(* PLC project testproj, Beckhoff Automation GmbH TwinCAT PLC Control 3.5.20.50 *)
(* stored: creationDateTime 2025-07-01T11:02:16.1300929, modificationDateTime 2025-07-01T11:02:16.1300929 *)

FUNCTION_BLOCK AnaMon
  VAR_INPUT
    WQC : BYTE;
    OSLevel : BYTE;
    V : REAL;
    VSclMin : REAL;
    VSclMax : REAL;
    VUnit : INT;
    VAHEn : BOOL;
    VWHEn : BOOL;
    VTHEn : BOOL;
    VTLEn : BOOL;
    VWLEn : BOOL;
    VALEn : BOOL;
  END_VAR
  VAR_OUTPUT
    VAHAct : BOOL;
    VWHAct : BOOL;
    VTHAct : BOOL;
    VTLAct : BOOL;
    VWLAct : BOOL;
    VALAct : BOOL;
  END_VAR
  VAR
    VAHLim : REAL;
    VWHLim : REAL;
    VTHLim : REAL;
    VTLLim : REAL;
    VWLLim : REAL;
    VALLim : REAL;
  END_VAR

            
                
// Copy MTP base variables to local temporaries (READ access)


VAHAct := vOut >= alarmHigh;
VWHAct := vOut >= warningHigh;
VTHAct := vOut >= toleranceHigh;
VTLAct := vOut <= toleranceLow;
VWLAct := vOut <= warningLow;
VALAct := vOut <= alarmLow;

// Copy local temporaries back to MTP base variables (WRITE access)
                
            
        
END_FUNCTION_BLOCK

FUNCTION_BLOCK BinMon
  VAR_INPUT
    WQC : BYTE;
    V : BOOL;
    VState0 : string;
    VState1 : string;
    OSLevel : BYTE;
    VFlutEn : BOOL;
  END_VAR
  VAR_OUTPUT
    VFlutAct : BOOL;
  END_VAR
  VAR
    VFlutTi : REAL;
    VFlutCnt : INT;
  END_VAR

            
                
// Copy MTP base variables to local temporaries (READ access)



// Copy local temporaries back to MTP base variables (WRITE access)
                
            
        
END_FUNCTION_BLOCK

FUNCTION_BLOCK LockView4
  VAR_INPUT
    WQC : BYTE;
    Logic : BOOL;
    In1En : BOOL;
    In1 : BOOL;
    In1QC : BYTE;
    In1Inv : BOOL;
    In1Txt : STRING;
    In2En : BOOL;
    In2 : BOOL;
    In2QC : BYTE;
    In2Inv : BOOL;
    In2Txt : STRING;
    In3En : BOOL;
    In3 : BOOL;
    In3QC : BYTE;
    In3Inv : BOOL;
    In3Txt : STRING;
    In4En : BOOL;
    In4 : BOOL;
    In4QC : BYTE;
    In4Inv : BOOL;
    In4Txt : STRING;
  END_VAR
  VAR_OUTPUT
    Out : BOOL;
    OutQC : STRING;
  END_VAR

            
                
// Copy MTP base variables to local temporaries (READ access)



// Copy local temporaries back to MTP base variables (WRITE access)
                
            
        
END_FUNCTION_BLOCK

FUNCTION_BLOCK MonAnaDrv
  VAR_INPUT
    StateChannel : BOOL;
    StateOffAut : BOOL;
    StateOpAut : BOOL;
    StateAutAut : BOOL;
    SrcChannel : BOOL;
    SrcManAut : BOOL;
    SrcIntAut : BOOL;
    PermEn : BOOL;
    Permit : BOOL;
    IntlEn : BOOL;
    Interlock : BOOL;
    ProtEn : BOOL;
    Protect : BOOL;
    WQC : BYTE;
    OSLevel : BYTE;
    SafePos : BOOL;
    FwdEn : BOOL;
    RevEn : BOOL;
    StopAut : BOOL;
    FwdAut : BOOL;
    RevAut : BOOL;
    RpmSclMin : REAL;
    RpmSclMax : REAL;
    RpmUnit : INT;
    RpmMin : REAL;
    RpmMax : REAL;
    RpmInt : REAL;
    RevFbkCalc : BOOL;
    RevFbk : BOOL;
    FwdFbkCalc : BOOL;
    FwdFbk : BOOL;
    RpmFbkCalc : BOOL;
    RpmFbk : REAL;
    Trip : BOOL;
    ResetAut : BOOL;
    MonSafePos : BOOL;
    MonStatTi : REAL;
    MonDynTi : REAL;
  END_VAR
  VAR_OUTPUT
    StateOpAct : BOOL;
    StateAutAct : BOOL;
    StateOffAct : BOOL;
    SrcIntAct : BOOL;
    SrcManAct : BOOL;
    SafePosAct : BOOL;
    FwdCtrl : BOOL;
    RevCtrl : BOOL;
    Rpm : REAL;
    MonStatErr : BOOL;
    MonDynErr : BOOL;
  END_VAR
  VAR
    StateOffOp : BOOL;
    StateOpOp : BOOL;
    StateAutOp : BOOL;
    SrcIntOp : BOOL;
    SrcManOp : BOOL;
    StopOp : BOOL;
    FwdOp : BOOL;
    RevOp : BOOL;
    RpmMan : REAL;
    RpmRbk : REAL;
    ResetOp : BOOL;
    MonEn : BOOL;
  END_VAR

            
                
// Copy MTP base variables to local temporaries (READ access)



// Copy local temporaries back to MTP base variables (WRITE access)
                
            
        
END_FUNCTION_BLOCK

FUNCTION_BLOCK MonAnaVlv
  VAR_INPUT
    StateChannel : BOOL;
    StateOffAut : BOOL;
    StateOpAut : BOOL;
    StateAutAut : BOOL;
    SrcChannel : BOOL;
    SrcManAut : BOOL;
    SrcIntAut : BOOL;
    PermEn : BOOL;
    Permit : BOOL;
    IntlEn : BOOL;
    Interlock : BOOL;
    ProtEn : BOOL;
    Protect : BOOL;
    WQC : BYTE;
    OSLevel : BYTE;
    SafePos : BOOL;
    SafePosEn : BOOL;
    OpenAut : BOOL;
    CloseAut : BOOL;
    PosSclMin : REAL;
    PosSclMax : REAL;
    PosUnit : INT;
    PosMin : REAL;
    PosMax : REAL;
    PosInt : REAL;
    OpenFbkCalc : BOOL;
    OpenFbk : BOOL;
    CloseFbkCalc : BOOL;
    CloseFbk : BOOL;
    PosFbkCalc : BOOL;
    PosFbk : REAL;
    ResetAut : BOOL;
  END_VAR
  VAR_OUTPUT
    StateOpAct : BOOL;
    StateAutAct : BOOL;
    StateOffAct : BOOL;
    SrcIntAct : BOOL;
    SrcManAct : BOOL;
    SafePosAct : BOOL;
    OpenAct : BOOL;
    CloseAct : BOOL;
    Pos : REAL;
  END_VAR
  VAR
    StateOffOp : BOOL;
    StateOpOp : BOOL;
    StateAutOp : BOOL;
    SrcIntOp : BOOL;
    SrcManOp : BOOL;
    OpenOp : BOOL;
    CloseOp : BOOL;
    PosMan : REAL;
    PosRbk : REAL;
    ResetOp : BOOL;
  END_VAR

            
                
// Copy MTP base variables to local temporaries (READ access)



// Copy local temporaries back to MTP base variables (WRITE access)
                
            
        
END_FUNCTION_BLOCK

FUNCTION_BLOCK MonBinDrv
  VAR_INPUT
    StateChannel : BOOL;
    StateOffAut : BOOL;
    StateOpAut : BOOL;
    StateAutAut : BOOL;
    PermEn : BOOL;
    Permit : BOOL;
    IntlEn : BOOL;
    Interlock : BOOL;
    ProtEn : BOOL;
    Protect : BOOL;
    WQC : BYTE;
    OSLevel : BYTE;
    SafePos : BOOL;
    FwdEn : BOOL;
    RevEn : BOOL;
    StopAut : BOOL;
    FwdAut : BOOL;
    RevAut : BOOL;
    RevFbkCalc : BOOL;
    RevFbk : BOOL;
    FwdFbkCalc : BOOL;
    FwdFbk : BOOL;
    Trip : BOOL;
    ResetAut : BOOL;
    MonSafePos : BOOL;
    MonStatTi : REAL;
    MonDynTi : REAL;
  END_VAR
  VAR_OUTPUT
    StateOpAct : BOOL;
    StateAutAct : BOOL;
    StateOffAct : BOOL;
    SafePosAct : BOOL;
    FwdCtrl : BOOL;
    RevCtrl : BOOL;
    MonStatErr : BOOL;
    MonDynErr : BOOL;
  END_VAR
  VAR
    StateOffOp : BOOL;
    StateOpOp : BOOL;
    StateAutOp : BOOL;
    StopOp : BOOL;
    FwdOp : BOOL;
    RevOp : BOOL;
    ResetOp : BOOL;
    MonEn : BOOL;
  END_VAR

            
                
// Copy MTP base variables to local temporaries (READ access)



// Copy local temporaries back to MTP base variables (WRITE access)
                
            
        
END_FUNCTION_BLOCK

FUNCTION_BLOCK MonBinVlv
  VAR_INPUT
    StateChannel : BOOL;
    StateOffAut : BOOL;
    StateOpAut : BOOL;
    StateAutAut : BOOL;
    PermEn : BOOL;
    IntlEn : BOOL;
    ProtEn : BOOL;
    Permit : BOOL;
    Interlock : BOOL;
    Protect : BOOL;
    WQC : BYTE;
    OSLevel : BYTE;
    SafePos : BOOL;
    SafePosEn : BOOL;
    OpenAut : BOOL;
    CloseAut : BOOL;
    OpenFbkCalc : BOOL;
    CloseFbkCalc : BOOL;
    OpenFbk : BOOL;
    CloseFbk : BOOL;
    MonSafePos : BOOL;
    MonStatTi : REAL;
    MonDynTi : REAL;
    ResetAut : BOOL;
  END_VAR
  VAR_OUTPUT
    StateOpAct : BOOL;
    StateAutAct : BOOL;
    StateOffAct : BOOL;
    SafePosAct : BOOL;
    Ctrl : BOOL;
    MonStatErr : BOOL;
    MonDynErr : BOOL;
    OperationMode : INT;
  END_VAR
  VAR
    StateOffOp : BOOL;
    StateOpOp : BOOL;
    StateAutOp : BOOL;
    OpenOp : BOOL;
    CloseOp : BOOL;
    ResetOp : BOOL;
    MonEn : BOOL;
    OpenedState : BOOL;
    ClosedState : BOOL;
  END_VAR

            
                
// Copy MTP base variables to local temporaries (READ access)



// Copy local temporaries back to MTP base variables (WRITE access)
                
            
        
END_FUNCTION_BLOCK

FUNCTION_BLOCK PIDCtrl
  VAR_INPUT
    StateChannel : BOOL;
    StateOffAut : BOOL;
    StateOpAut : BOOL;
    StateAutAut : BOOL;
    SrcChannel : BOOL;
    SrcManAut : BOOL;
    SrcIntAut : BOOL;
    WQC : BYTE;
    OSLevel : BYTE;
    PV : REAL;
    PVSclMin : REAL;
    PVSclMax : REAL;
    PVUnit : INT;
    SPInt : REAL;
    SPSclMin : REAL;
    SPSclMax : REAL;
    SPUnit : INT;
    SPIntMin : REAL;
    SPIntMax : REAL;
    SPManMin : REAL;
    SPManMax : REAL;
    MVMin : REAL;
    MVMax : REAL;
    MVUnit : INT;
    MVSclMin : REAL;
    MVSclMax : REAL;
    P : REAL;
    Ti : REAL;
    Td : REAL;
  END_VAR
  VAR_OUTPUT
    StateOpAct : BOOL;
    StateAutAct : BOOL;
    StateOffAct : BOOL;
    SrcIntAct : BOOL;
    SrcManAct : BOOL;
    SP : REAL;
    MV : REAL;
  END_VAR
  VAR
    StateOffOp : BOOL;
    StateOpOp : BOOL;
    StateAutOp : BOOL;
    SrcIntOp : BOOL;
    SrcManOp : BOOL;
    SPMan : REAL;
    MVMan : REAL;
  END_VAR

            
                
// Copy MTP base variables to local temporaries (READ access)



// Copy local temporaries back to MTP base variables (WRITE access)
                
            
        
END_FUNCTION_BLOCK

FUNCTION_BLOCK AnalogMeasurement
  VAR_IN_OUT
    MTPBase : AnaMon;
  END_VAR
  VAR_INPUT
    id : INT;
    rawValue : WORD;
    valueUnit : INT;
    scaleMin : REAL;
    scaleMax : REAL;
    alarmHigh : REAL;
    warningHigh : REAL;
    toleranceHigh : REAL;
    toleranceLow : REAL;
    warningLow : REAL;
    alarmLow : REAL;
    alarmHighEn : BOOL;
    warningHighEn : BOOL;
    toleranceHighEn : BOOL;
    toleranceLowEn : BOOL;
    warningLowEn : BOOL;
    alarmLowEn : BOOL;
    deadband : REAL;
    externalFault : BOOL;
  END_VAR
  VAR_OUTPUT
    vOut : REAL;
    error : BOOL;
    alarmHighStatus : BOOL;
    warningHighStatus : BOOL;
    toleranceHighStatus : BOOL;
    toleranceLowStatus : BOOL;
    warningLowStatus : BOOL;
    alarmLowStatus : BOOL;
  END_VAR
  VAR
    WQC : BYTE;
    OSLevel : BYTE;
    V : REAL;
    VSclMin : REAL;
    VSclMax : REAL;
    VUnit : INT;
    VAHEn : BOOL;
    VWHEn : BOOL;
    VTHEn : BOOL;
    VTLEn : BOOL;
    VWLEn : BOOL;
    VALEn : BOOL;
    VAHLim : REAL;
    VWHLim : REAL;
    VTHLim : REAL;
    VTLLim : REAL;
    VWLLim : REAL;
    VALLim : REAL;
  END_VAR

            
                
// Copy MTP base variables to local temporaries (READ access)
V := MTPBase.V;
VSclMin := MTPBase.VSclMin;
VSclMax := MTPBase.VSclMax;
VAHLim := MTPBase.VAHLim;
VWHLim := MTPBase.VWHLim;
VTHLim := MTPBase.VTHLim;
VTLLim := MTPBase.VTLLim;
VWLLim := MTPBase.VWLLim;
VALLim := MTPBase.VALLim;


WQC := 16#FF;
OSLevel := 16#00;
V := VSclMin + (WORD_TO_REAL(rawValue) / 27648.0) * (VSclMax - VSclMin);
vOut := V;
VSclMin := scaleMin;
VSclMax := scaleMax;
VUnit := valueUnit;
VAHEn := alarmHighEn;
VWHEn := warningHighEn;
VTHEn := toleranceHighEn;
VTLEn := toleranceLowEn;
VWLEn := warningLowEn;
VALEn := alarmLowEn;

// Copy local temporaries back to MTP base variables (WRITE access)
MTPBase.WQC := WQC;
MTPBase.OSLevel := OSLevel;
MTPBase.V := V;
MTPBase.VSclMin := VSclMin;
MTPBase.VSclMax := VSclMax;
MTPBase.VUnit := VUnit;
MTPBase.VAHEn := VAHEn;
MTPBase.VWHEn := VWHEn;
MTPBase.VTHEn := VTHEn;
MTPBase.VTLEn := VTLEn;
MTPBase.VWLEn := VWLEn;
MTPBase.VALEn := VALEn;
                
            
        
END_FUNCTION_BLOCK

FUNCTION_BLOCK AnalogValve
  VAR_IN_OUT
    MTPBase : MonAnaVlv;
  END_VAR
  VAR_INPUT
    id : INT;
    activateManualSource : BOOL;
    activateDynamicSource : BOOL;
    activateFixedSource : BOOL;
    dynamicSource : REAL;
    fixedSource : REAL;
    feedbackPosition : WORD;
    scaleMin : REAL;
    scaleMax : REAL;
    feedbackOpen : BOOL;
    feedbackClose : BOOL;
    hasFbOpen : BOOL;
    hasFbClose : BOOL;
    safeOpen : BOOL;
    enableSafePos : BOOL;
    simulate : BOOL;
    simulateDelay : REAL;
    interlockIn : BOOL;
    permitIn : BOOL;
    protectIn : BOOL;
    reset : BOOL;
  END_VAR
  VAR_OUTPUT
    positionOutDevice : WORD;
    positionOut : REAL;
    remote : BOOL;
    operatorMode : BOOL;
    automaticMode : BOOL;
    offlineMode : BOOL;
    error : BOOL;
    opened : BOOL;
    closed : BOOL;
    programSelectsSource : BOOL;
    operatorSelectsSource : BOOL;
    manualSourceAct : BOOL;
    internalSourceAct : BOOL;
    dynamicSourceAct : BOOL;
    fixedSourceAct : BOOL;
  END_VAR
  VAR
    fbOpenSimulated : BOOL;
    fbCloseSimulated : BOOL;
    selectedPosition : REAL;
    DelayTimer1 : TON;
    DelayTimer2 : TON;
    StateChannel : BOOL;
    StateOpAct : BOOL;
    StateAutAct : BOOL;
    StateOffAct : BOOL;
    SrcChannel : BOOL;
    SrcManAut : BOOL;
    SrcIntAut : BOOL;
    SrcIntAct : BOOL;
    SrcManAct : BOOL;
    PermEn : BOOL;
    Permit : BOOL;
    IntlEn : BOOL;
    Interlock : BOOL;
    ProtEn : BOOL;
    Protect : BOOL;
    WQC : BYTE;
    OSLevel : BYTE;
    SafePos : BOOL;
    SafePosEn : BOOL;
    OpenAut : BOOL;
    CloseAut : BOOL;
    PosSclMin : REAL;
    PosSclMax : REAL;
    PosUnit : INT;
    PosMin : REAL;
    PosMax : REAL;
    PosInt : REAL;
    PosMan : REAL;
    Pos : REAL;
    OpenFbkCalc : BOOL;
    OpenFbk : BOOL;
    CloseFbkCalc : BOOL;
    CloseFbk : BOOL;
    PosFbkCalc : BOOL;
    PosFbk : REAL;
    ResetAut : BOOL;
  END_VAR

            
                
// Copy MTP base variables to local temporaries (READ access)
StateChannel := MTPBase.StateChannel;
StateOpAct := MTPBase.StateOpAct;
StateAutAct := MTPBase.StateAutAct;
StateOffAct := MTPBase.StateOffAct;
SrcChannel := MTPBase.SrcChannel;
SrcIntAct := MTPBase.SrcIntAct;
SrcManAct := MTPBase.SrcManAct;
OpenAut := MTPBase.OpenAut;
PosSclMin := MTPBase.PosSclMin;
PosSclMax := MTPBase.PosSclMax;
PosInt := MTPBase.PosInt;
PosMan := MTPBase.PosMan;
Pos := MTPBase.Pos;
OpenFbkCalc := MTPBase.OpenFbkCalc;
OpenFbk := MTPBase.OpenFbk;
CloseFbkCalc := MTPBase.CloseFbkCalc;
CloseFbk := MTPBase.CloseFbk;


WQC := 16#FF;
OSLevel := 16#00;
remote := StateChannel;
operatorMode := StateOpAct;
automaticMode := StateAutAct;
offlineMode := StateOffAct;
programSelectsSource := SrcChannel;
operatorSelectsSource := NOT SrcChannel;
internalSourceAct := SrcIntAct;
manualSourceAct := SrcManAct;
SrcManAut := activateManualSource;
SrcIntAut := activateDynamicSource OR activateFixedSource;
IF activateFixedSource THEN
    fixedSourceAct := TRUE;
END_IF;
IF activateDynamicSource THEN
    fixedSourceAct := FALSE;
END_IF;
dynamicSourceAct := NOT fixedSourceAct;
PermEn := True;
IntlEn := True;
ProtEn := True;
Permit := permitIn;
Interlock := NOT interlockIn;
Protect := NOT protectIn;
SafePos := safeOpen;
SafePosEn := enableSafePos;
selectedPosition := (PosInt * BOOL_TO_REAL(SrcIntAct)) + (PosMan * BOOL_TO_REAL(SrcManAct));
OpenAut := selectedPosition > 0;
CloseAut := NOT OpenAut;
OpenFbkCalc := simulate OR NOT hasFbOpen;
CloseFbkCalc := simulate OR NOT hasFbClose;
PosFbkCalc := simulate;
DelayTimer1(IN:= OpenFbkCalc AND OpenAut, PT:= REAL_TO_TIME(simulateDelay * 1000));
fbOpenSimulated := DelayTimer1.Q;
DelayTimer2(IN:= CloseFbkCalc AND NOT OpenAut, PT:= REAL_TO_TIME(simulateDelay * 1000));
fbCloseSimulated := DelayTimer2.Q;
OpenFbk := (feedbackOpen AND NOT OpenFbkCalc) OR (fbOpenSimulated AND OpenFbkCalc);
CloseFbk := (feedbackClose AND NOT CloseFbkCalc) OR (fbCloseSimulated AND CloseFbkCalc);
opened := OpenFbk;
closed := CloseFbk;
ResetAut := reset;
PosSclMin := scaleMin;
PosSclMax := scaleMax;
PosUnit := 0;
PosMin := PosSclMin;
PosMax := PosSclMax;
PosInt := (dynamicSource * BOOL_TO_REAL(dynamicSourceAct)) + (fixedSource * BOOL_TO_REAL(fixedSourceAct));
PosFbk := (positionOut * BOOL_TO_REAL(simulate)) + (feedbackPosition * BOOL_TO_REAL(simulate));
positionOut := Pos;
reset := False;
activateManualSource := False;
activateDynamicSource := False;
activateFixedSource := False;

// Copy local temporaries back to MTP base variables (WRITE access)
MTPBase.SrcManAut := SrcManAut;
MTPBase.SrcIntAut := SrcIntAut;
MTPBase.PermEn := PermEn;
MTPBase.Permit := Permit;
MTPBase.IntlEn := IntlEn;
MTPBase.Interlock := Interlock;
MTPBase.ProtEn := ProtEn;
MTPBase.Protect := Protect;
MTPBase.WQC := WQC;
MTPBase.OSLevel := OSLevel;
MTPBase.SafePos := SafePos;
MTPBase.SafePosEn := SafePosEn;
MTPBase.OpenAut := OpenAut;
MTPBase.CloseAut := CloseAut;
MTPBase.PosSclMin := PosSclMin;
MTPBase.PosSclMax := PosSclMax;
MTPBase.PosUnit := PosUnit;
MTPBase.PosMin := PosMin;
MTPBase.PosMax := PosMax;
MTPBase.PosInt := PosInt;
MTPBase.OpenFbkCalc := OpenFbkCalc;
MTPBase.OpenFbk := OpenFbk;
MTPBase.CloseFbkCalc := CloseFbkCalc;
MTPBase.CloseFbk := CloseFbk;
MTPBase.PosFbkCalc := PosFbkCalc;
MTPBase.PosFbk := PosFbk;
MTPBase.ResetAut := ResetAut;
                
            
        
END_FUNCTION_BLOCK

FUNCTION_BLOCK DigitalMeasurement
  VAR_IN_OUT
    MTPBase : BinMon;
  END_VAR
  VAR_INPUT
    id : INT;
    value : BOOL;
  END_VAR
  VAR_OUTPUT
    valueOut : BOOL;
    risingEdge : BOOL;
    fallingEdge : BOOL;
  END_VAR
  VAR
    lastValue : BOOL;
    WQC : BYTE;
    V : BOOL;
    VState0 : string;
    VState1 : string;
    OSLevel : BYTE;
    VFlutEn : BOOL;
  END_VAR

            
                
// Copy MTP base variables to local temporaries (READ access)


WQC := 16#FF;
OSLevel := 16#00;
V := value;
VState0 := 'False';
VState1 := 'True';
VFlutEn := False;
risingEdge := value <> lastValue and value = True;
fallingEdge := value <> lastValue and value = False;
lastValue := value;

// Copy local temporaries back to MTP base variables (WRITE access)
MTPBase.WQC := WQC;
MTPBase.V := V;
MTPBase.VState0 := VState0;
MTPBase.VState1 := VState1;
MTPBase.OSLevel := OSLevel;
MTPBase.VFlutEn := VFlutEn;
                
            
        
END_FUNCTION_BLOCK

FUNCTION_BLOCK Interlock4

            
                
// Copy MTP base variables to local temporaries (READ access)



// Copy local temporaries back to MTP base variables (WRITE access)
                
            
        
END_FUNCTION_BLOCK

FUNCTION_BLOCK PIDController
  VAR_IN_OUT
    MTPBase : PIDCtrl;
  END_VAR
  VAR_INPUT
    id : INT;
    activateManualSP : BOOL;
    activateDynamicSP : BOOL;
    activateFixedSP : BOOL;
    dynamicSP : REAL;
    fixedSP : REAL;
    rawValue : WORD;
    valueUnit : INT;
    manipulatedValueUnit : INT;
    scaleMin : REAL;
    scaleMax : REAL;
    scaleMinMV : REAL;
    scaleMaxMV : REAL;
    proportional : REAL;
    integration : REAL;
    derivation : REAL;
    alarmHigh : REAL;
    warningHigh : REAL;
    toleranceHigh : REAL;
    toleranceLow : REAL;
    warningLow : REAL;
    alarmLow : REAL;
    alarmHighEn : BOOL;
    warningHighEn : BOOL;
    toleranceHighEn : BOOL;
    toleranceLowEn : BOOL;
    warningLowEn : BOOL;
    alarmLowEn : BOOL;
    deadband : REAL;
    externalFault : BOOL;
  END_VAR
  VAR_OUTPUT
    setpointOut : REAL;
    valueOut : REAL;
    manipulatedValue : REAL;
    remote : BOOL;
    operatorMode : BOOL;
    automaticMode : BOOL;
    offlineMode : BOOL;
    error : BOOL;
    alarmHighStatus : BOOL;
    warningHighStatus : BOOL;
    toleranceHighStatus : BOOL;
    toleranceLowStatus : BOOL;
    warningLowStatus : BOOL;
    alarmLowStatus : BOOL;
    programSelectsSP : BOOL;
    operatorSelectsSP : BOOL;
    manualSPAct : BOOL;
    internalSPAct : BOOL;
    dynamicSPAct : BOOL;
    fixedSPAct : BOOL;
  END_VAR
  VAR
    StateChannel : BOOL;
    StateOpAct : BOOL;
    StateAutAct : BOOL;
    StateOffAct : BOOL;
    SrcChannel : BOOL;
    SrcManAut : BOOL;
    SrcIntAut : BOOL;
    SrcIntAct : BOOL;
    SrcManAct : BOOL;
    WQC : BYTE;
    OSLevel : BYTE;
    PV : REAL;
    PVSclMin : REAL;
    PVSclMax : REAL;
    PVUnit : INT;
    SPInt : REAL;
    SPSclMin : REAL;
    SPSclMax : REAL;
    SPUnit : INT;
    SPIntMin : REAL;
    SPIntMax : REAL;
    SPManMin : REAL;
    SPManMax : REAL;
    SP : REAL;
    MV : REAL;
    MVMin : REAL;
    MVMax : REAL;
    MVUnit : INT;
    MVSclMin : REAL;
    MVSclMax : REAL;
    P : REAL;
    Ti : REAL;
    Td : REAL;
  END_VAR

            
                
// Copy MTP base variables to local temporaries (READ access)
StateChannel := MTPBase.StateChannel;
StateOpAct := MTPBase.StateOpAct;
StateAutAct := MTPBase.StateAutAct;
StateOffAct := MTPBase.StateOffAct;
SrcChannel := MTPBase.SrcChannel;
SrcIntAct := MTPBase.SrcIntAct;
SrcManAct := MTPBase.SrcManAct;
PV := MTPBase.PV;
SP := MTPBase.SP;
MV := MTPBase.MV;
P := MTPBase.P;
Ti := MTPBase.Ti;
Td := MTPBase.Td;


WQC := 16#FF;
OSLevel := 16#00;
remote := StateChannel;
operatorMode := StateOpAct;
automaticMode := StateAutAct;
offlineMode := StateOffAct;
programSelectsSP := SrcChannel;
operatorSelectsSP := NOT SrcChannel;
internalSPAct := SrcIntAct;
manualSPAct := SrcManAct;
SrcManAut := activateManualSP;
SrcIntAut := activateDynamicSP OR activateFixedSP;
IF activateFixedSP THEN
    fixedSPAct := TRUE;
END_IF;
IF activateDynamicSP THEN
    fixedSPAct := FALSE;
END_IF;
dynamicSPAct := NOT fixedSPAct;
PV := scaleMin + (WORD_TO_REAL(rawValue) / 27648.0) * (scaleMax - scaleMin);
valueOut := PV;
PVSclMin := scaleMin;
PVSclMax := scaleMax;
PVUnit := valueUnit;
SPInt := (dynamicSP * BOOL_TO_REAL(dynamicSPAct)) + (fixedSP * BOOL_TO_REAL(fixedSPAct));
SPSclMin := scaleMin;
SPSclMax := scaleMax;
SPUnit := valueUnit;
SPIntMin := scaleMin;
SPIntMax := scaleMax;
SPManMin := scaleMin;
SPManMax := scaleMax;
setpointOut := SP;
manipulatedValue := MV;
MVMin := scaleMinMV;
MVMax := scaleMaxMV;
MVUnit := manipulatedValueUnit;
MVSclMin := scaleMinMV;
MVSclMax := scaleMaxMV;
activateManualSP := False;
activateDynamicSP := False;
activateFixedSP := False;

// Copy local temporaries back to MTP base variables (WRITE access)
MTPBase.SrcManAut := SrcManAut;
MTPBase.SrcIntAut := SrcIntAut;
MTPBase.WQC := WQC;
MTPBase.OSLevel := OSLevel;
MTPBase.PV := PV;
MTPBase.PVSclMin := PVSclMin;
MTPBase.PVSclMax := PVSclMax;
MTPBase.PVUnit := PVUnit;
MTPBase.SPInt := SPInt;
MTPBase.SPSclMin := SPSclMin;
MTPBase.SPSclMax := SPSclMax;
MTPBase.SPUnit := SPUnit;
MTPBase.SPIntMin := SPIntMin;
MTPBase.SPIntMax := SPIntMax;
MTPBase.SPManMin := SPManMin;
MTPBase.SPManMax := SPManMax;
MTPBase.MVMin := MVMin;
MTPBase.MVMax := MVMax;
MTPBase.MVUnit := MVUnit;
MTPBase.MVSclMin := MVSclMin;
MTPBase.MVSclMax := MVSclMax;
                
            
        
END_FUNCTION_BLOCK

FUNCTION_BLOCK ReversingMotor
  VAR_IN_OUT
    MTPBase : MonBinDrv;
  END_VAR
  VAR_INPUT
    id : INT;
    forward : BOOL;
    reverse : BOOL;
    stop : BOOL;
    forwardFeedback : BOOL;
    reverseFeedback : BOOL;
    hasFwdFeedback : BOOL;
    hasRevFeedback : BOOL;
    enableForward : BOOL;
    enableReverse : BOOL;
    driveTrip : BOOL;
    safeHold : BOOL;
    monitor : BOOL;
    staticTimeout : REAL;
    dynamicTimeout : REAL;
    simulate : BOOL;
    simulateDelay : REAL;
    interlockIn : BOOL;
    permitIn : BOOL;
    protectIn : BOOL;
    reset : BOOL;
  END_VAR
  VAR_OUTPUT
    fwdCommand : BOOL;
    revCommand : BOOL;
    forwardActive : BOOL;
    reverseActive : BOOL;
    stopped : BOOL;
    remote : BOOL;
    operatorMode : BOOL;
    automaticMode : BOOL;
    offlineMode : BOOL;
  END_VAR
  VAR
    fwdFbkSimulated : BOOL;
    revFbkSimulated : BOOL;
    DelayTimer1 : TON;
    DelayTimer2 : TON;
    StateChannel : BOOL;
    StateOpAct : BOOL;
    StateAutAct : BOOL;
    StateOffAct : BOOL;
    PermEn : BOOL;
    Permit : BOOL;
    IntlEn : BOOL;
    Interlock : BOOL;
    ProtEn : BOOL;
    Protect : BOOL;
    WQC : BYTE;
    OSLevel : BYTE;
    SafePos : BOOL;
    FwdEn : BOOL;
    RevEn : BOOL;
    StopAut : BOOL;
    FwdAut : BOOL;
    RevAut : BOOL;
    FwdCtrl : BOOL;
    RevCtrl : BOOL;
    RevFbkCalc : BOOL;
    RevFbk : BOOL;
    FwdFbkCalc : BOOL;
    FwdFbk : BOOL;
    Trip : BOOL;
    ResetAut : BOOL;
    MonSafePos : BOOL;
    MonStatTi : REAL;
    MonDynTi : REAL;
  END_VAR

            
                
// Copy MTP base variables to local temporaries (READ access)
StateChannel := MTPBase.StateChannel;
StateOpAct := MTPBase.StateOpAct;
StateAutAct := MTPBase.StateAutAct;
StateOffAct := MTPBase.StateOffAct;
FwdCtrl := MTPBase.FwdCtrl;
RevCtrl := MTPBase.RevCtrl;
RevFbkCalc := MTPBase.RevFbkCalc;
RevFbk := MTPBase.RevFbk;
FwdFbkCalc := MTPBase.FwdFbkCalc;
FwdFbk := MTPBase.FwdFbk;


WQC := 16#FF;
OSLevel := 16#00;
remote := StateChannel;
operatorMode := StateOpAct;
automaticMode := StateAutAct;
offlineMode := StateOffAct;
PermEn := True;
IntlEn := True;
ProtEn := True;
Permit := permitIn;
Interlock := NOT interlockIn;
Protect := NOT protectIn;
SafePos := false;
FwdEn := enableForward;
RevEn := enableReverse;
StopAut := (NOT forward AND NOT reverse) OR stop;
IF forward AND NOT stop THEN
    FwdAut := TRUE;
END_IF;
IF stop THEN
    FwdAut := FALSE;
END_IF;
IF reverse AND NOT stop THEN
    RevAut := TRUE;
END_IF;
IF stop THEN
    RevAut := FALSE;
END_IF;
fwdCommand := FwdCtrl;
revCommand := RevCtrl;
FwdFbkCalc := simulate OR NOT hasFwdFeedback;
RevFbkCalc := simulate OR NOT hasRevFeedback;
DelayTimer1(IN:= FwdFbkCalc AND fwdCommand, PT:= REAL_TO_TIME(simulateDelay * 1000));
fwdFbkSimulated := DelayTimer1.Q;
DelayTimer2(IN:= RevFbkCalc AND revCommand, PT:= REAL_TO_TIME(simulateDelay * 1000));
revFbkSimulated := DelayTimer2.Q;
FwdFbk := (forwardFeedback AND NOT FwdFbkCalc) OR (fwdFbkSimulated AND FwdFbkCalc);
RevFbk := (reverseFeedback AND NOT RevFbkCalc) OR (revFbkSimulated AND RevFbkCalc);
forwardActive := FwdFbk;
reverseActive := RevFbk;
stopped := NOT FwdFbk AND NOT RevFbk;
Trip := NOT driveTrip;
ResetAut := reset;
MonSafePos := safeHold;
MonStatTi := staticTimeout;
MonDynTi := dynamicTimeout;
reset := False;
stop := False;

// Copy local temporaries back to MTP base variables (WRITE access)
MTPBase.PermEn := PermEn;
MTPBase.Permit := Permit;
MTPBase.IntlEn := IntlEn;
MTPBase.Interlock := Interlock;
MTPBase.ProtEn := ProtEn;
MTPBase.Protect := Protect;
MTPBase.WQC := WQC;
MTPBase.OSLevel := OSLevel;
MTPBase.SafePos := SafePos;
MTPBase.FwdEn := FwdEn;
MTPBase.RevEn := RevEn;
MTPBase.StopAut := StopAut;
MTPBase.FwdAut := FwdAut;
MTPBase.RevAut := RevAut;
MTPBase.RevFbkCalc := RevFbkCalc;
MTPBase.RevFbk := RevFbk;
MTPBase.FwdFbkCalc := FwdFbkCalc;
MTPBase.FwdFbk := FwdFbk;
MTPBase.Trip := Trip;
MTPBase.ResetAut := ResetAut;
MTPBase.MonSafePos := MonSafePos;
MTPBase.MonStatTi := MonStatTi;
MTPBase.MonDynTi := MonDynTi;
                
            
        
END_FUNCTION_BLOCK

FUNCTION_BLOCK SolenoidValve
  VAR_IN_OUT
    MTPBase : MonBinVlv;
  END_VAR
  VAR_INPUT
    id : INT;
    open : BOOL;
    close : BOOL;
    outsideOpen : BOOL;
    outsideClose : BOOL;
    feedbackOpen : BOOL;
    feedbackClose : BOOL;
    hasFbOpen : BOOL;
    hasFbClose : BOOL;
    safeOpen : BOOL;
    safeHold : BOOL;
    monitor : BOOL;
    staticTimeout : REAL;
    dynamicTimeout : REAL;
    simulate : BOOL;
    simulateDelay : REAL;
    interlockIn : BOOL;
    permitIn : BOOL;
    protectIn : BOOL;
    reset : BOOL;
    externalFault : BOOL;
    surpressAlarms : BOOL;
    setAuto : BOOL;
    setManual : BOOL;
    setOutside : BOOL;
  END_VAR
  VAR_OUTPUT
    openCommand : BOOL;
    pulseOpen : BOOL;
    pulseClose : BOOL;
    remote : BOOL;
    operatorMode : BOOL;
    automaticMode : BOOL;
    offlineMode : BOOL;
    outside : BOOL;
    error : BOOL;
    opened : BOOL;
    closed : BOOL;
    forceActive : BOOL;
    surpressed : BOOL;
  END_VAR
  VAR
    fbOpenSimulated : BOOL;
    fbCloseSimulated : BOOL;
    DelayTimer1 : TON;
    DelayTimer2 : TON;
    StateChannel : BOOL;
    StateOpAct : BOOL;
    StateAutAct : BOOL;
    StateOffAct : BOOL;
    PermEn : BOOL;
    IntlEn : BOOL;
    ProtEn : BOOL;
    Permit : BOOL;
    Interlock : BOOL;
    Protect : BOOL;
    WQC : BYTE;
    SafePos : BOOL;
    SafePosEn : BOOL;
    OpenAut : BOOL;
    CloseAut : BOOL;
    Ctrl : BOOL;
    OpenFbkCalc : BOOL;
    CloseFbkCalc : BOOL;
    OpenFbk : BOOL;
    CloseFbk : BOOL;
    MonSafePos : BOOL;
    MonStatTi : REAL;
    MonDynTi : REAL;
    ResetAut : BOOL;
    MonEn : BOOL;
  END_VAR

            
                
// Copy MTP base variables to local temporaries (READ access)
StateChannel := MTPBase.StateChannel;
StateOpAct := MTPBase.StateOpAct;
StateAutAct := MTPBase.StateAutAct;
StateOffAct := MTPBase.StateOffAct;
Ctrl := MTPBase.Ctrl;
OpenFbkCalc := MTPBase.OpenFbkCalc;
CloseFbkCalc := MTPBase.CloseFbkCalc;
OpenFbk := MTPBase.OpenFbk;
CloseFbk := MTPBase.CloseFbk;


WQC := 16#FF;
remote := StateChannel;
operatorMode := StateOpAct;
automaticMode := StateAutAct;
offlineMode := StateOffAct;
PermEn := True;
IntlEn := True;
ProtEn := True;
Permit := permitIn;
Interlock := NOT interlockIn;
Protect := NOT protectIn;
SafePos := safeOpen;
MonSafePos := safeOpen;
SafePosEn := safeHold;
OpenAut := open;
CloseAut := close;
OpenFbkCalc := simulate OR NOT hasFbOpen;
CloseFbkCalc := simulate OR NOT hasFbClose;
DelayTimer1(IN:= OpenFbkCalc AND Ctrl, PT:= REAL_TO_TIME(simulateDelay * 1000));
fbOpenSimulated := DelayTimer1.Q;
DelayTimer2(IN:= CloseFbkCalc AND NOT Ctrl, PT:= REAL_TO_TIME(simulateDelay * 1000));
fbCloseSimulated := DelayTimer2.Q;
OpenFbk := (feedbackOpen AND NOT OpenFbkCalc) OR (fbOpenSimulated AND OpenFbkCalc);
CloseFbk := (feedbackClose AND NOT CloseFbkCalc) OR (fbCloseSimulated AND CloseFbkCalc);
opened := Ctrl AND OpenFbk;
closed := NOT Ctrl AND CloseFbk;
ResetAut := reset;
MonEn := monitor;
MonStatTi := staticTimeout;
MonDynTi := dynamicTimeout;
reset := False;

// Copy local temporaries back to MTP base variables (WRITE access)
MTPBase.PermEn := PermEn;
MTPBase.IntlEn := IntlEn;
MTPBase.ProtEn := ProtEn;
MTPBase.Permit := Permit;
MTPBase.Interlock := Interlock;
MTPBase.Protect := Protect;
MTPBase.WQC := WQC;
MTPBase.SafePos := SafePos;
MTPBase.SafePosEn := SafePosEn;
MTPBase.OpenAut := OpenAut;
MTPBase.CloseAut := CloseAut;
MTPBase.OpenFbkCalc := OpenFbkCalc;
MTPBase.CloseFbkCalc := CloseFbkCalc;
MTPBase.OpenFbk := OpenFbk;
MTPBase.CloseFbk := CloseFbk;
MTPBase.MonSafePos := MonSafePos;
MTPBase.MonStatTi := MonStatTi;
MTPBase.MonDynTi := MonDynTi;
MTPBase.ResetAut := ResetAut;
MTPBase.MonEn := MonEn;
                
            
        
END_FUNCTION_BLOCK

FUNCTION_BLOCK VFD
  VAR_IN_OUT
    MTPBase : MonAnaDrv;
  END_VAR
  VAR_INPUT
    id : INT;
    forward : BOOL;
    reverse : BOOL;
    speed : REAL;
    speedUnit : INT;
    speedMin : REAL;
    speedMax : REAL;
    forwardFeedback : BOOL;
    reverseFeedback : BOOL;
    speedFeedback : WORD;
    speedScaleMin : REAL;
    speedScaleMax : REAL;
    hasFwdFeedback : BOOL;
    hasRevFeedback : BOOL;
    enableForward : BOOL;
    enableReverse : BOOL;
    trip : BOOL;
    safeHold : BOOL;
    monitor : BOOL;
    staticTimeout : REAL;
    dynamicTimeout : REAL;
    simulate : BOOL;
    simulateDelay : REAL;
    interlockIn : BOOL;
    permitIn : BOOL;
    protectIn : BOOL;
    reset : BOOL;
  END_VAR
  VAR_OUTPUT
    fwdCommand : BOOL;
    revCommand : BOOL;
    forwardActive : BOOL;
    reverseActive : BOOL;
    actualSpeed : REAL;
    remote : BOOL;
    operatorMode : BOOL;
    automaticMode : BOOL;
    offlineMode : BOOL;
    remoteSource : BOOL;
    internalSourceAct : BOOL;
    manualSourceAct : BOOL;
  END_VAR
  VAR
    fwdFbkSimulated : BOOL;
    revFbkSimulated : BOOL;
    DelayTimer1 : TON;
    DelayTimer2 : TON;
    StateChannel : BOOL;
    StateOpAct : BOOL;
    StateAutAct : BOOL;
    StateOffAct : BOOL;
    SrcChannel : BOOL;
    SrcIntAct : BOOL;
    SrcManAct : BOOL;
    PermEn : BOOL;
    Permit : BOOL;
    IntlEn : BOOL;
    Interlock : BOOL;
    ProtEn : BOOL;
    Protect : BOOL;
    WQC : BYTE;
    OSLevel : BYTE;
    SafePos : BOOL;
    FwdAut : BOOL;
    RevAut : BOOL;
    FwdCtrl : BOOL;
    RevCtrl : BOOL;
    RpmSclMin : REAL;
    RpmSclMax : REAL;
    RpmUnit : INT;
    RpmMin : REAL;
    RpmMax : REAL;
    RpmRbk : REAL;
    Rpm : REAL;
    RevFbkCalc : BOOL;
    RevFbk : BOOL;
    FwdFbkCalc : BOOL;
    FwdFbk : BOOL;
    Trip : BOOL;
    ResetAut : BOOL;
    MonSafePos : BOOL;
    MonStatTi : REAL;
    MonDynTi : REAL;
  END_VAR

            
                
// Copy MTP base variables to local temporaries (READ access)
StateChannel := MTPBase.StateChannel;
StateOpAct := MTPBase.StateOpAct;
StateAutAct := MTPBase.StateAutAct;
StateOffAct := MTPBase.StateOffAct;
SrcChannel := MTPBase.SrcChannel;
SrcIntAct := MTPBase.SrcIntAct;
SrcManAct := MTPBase.SrcManAct;
FwdCtrl := MTPBase.FwdCtrl;
RevCtrl := MTPBase.RevCtrl;
Rpm := MTPBase.Rpm;
RevFbkCalc := MTPBase.RevFbkCalc;
FwdFbkCalc := MTPBase.FwdFbkCalc;


WQC := 16#FF;
OSLevel := 16#00;
remote := StateChannel;
operatorMode := StateOpAct;
automaticMode := StateAutAct;
offlineMode := StateOffAct;
remoteSource := SrcChannel;
internalSourceAct := SrcIntAct;
manualSourceAct := SrcManAct;
PermEn := True;
IntlEn := True;
ProtEn := True;
Permit := permitIn;
Interlock := NOT interlockIn;
Protect := NOT protectIn;
SafePos := False;
FwdAut := forward;
RevAut := reverse;
fwdCommand := FwdCtrl;
revCommand := RevCtrl;
FwdFbkCalc := simulate OR NOT hasFwdFeedback;
RevFbkCalc := simulate OR NOT hasRevFeedback;
DelayTimer1(IN:= (simulate OR NOT hasFwdFeedback) AND fwdCommand, PT:= REAL_TO_TIME(simulateDelay * 1000));
fwdFbkSimulated := DelayTimer1.Q;
DelayTimer2(IN:= (simulate OR NOT hasRevFeedback) AND NOT revCommand, PT:= REAL_TO_TIME(simulateDelay * 1000));
revFbkSimulated := DelayTimer2.Q;
FwdFbk := (forwardFeedback AND NOT FwdFbkCalc) OR (fwdFbkSimulated AND FwdFbkCalc);
RevFbk := (reverseFeedback AND NOT RevFbkCalc) OR (revFbkSimulated AND RevFbkCalc);
Trip := trip;
ResetAut := reset;
RpmSclMin := speedMin;
RpmSclMax := speedMax;
RpmUnit := speedUnit;
RpmMin := speedMin;
RpmMax := speedMax;
RpmRbk := speedFeedback;
actualSpeed := Rpm;
reset := False;
MonSafePos := safeHold;
MonStatTi := staticTimeout;
MonDynTi := dynamicTimeout;

// Copy local temporaries back to MTP base variables (WRITE access)
MTPBase.PermEn := PermEn;
MTPBase.Permit := Permit;
MTPBase.IntlEn := IntlEn;
MTPBase.Interlock := Interlock;
MTPBase.ProtEn := ProtEn;
MTPBase.Protect := Protect;
MTPBase.WQC := WQC;
MTPBase.OSLevel := OSLevel;
MTPBase.SafePos := SafePos;
MTPBase.FwdAut := FwdAut;
MTPBase.RevAut := RevAut;
MTPBase.RpmSclMin := RpmSclMin;
MTPBase.RpmSclMax := RpmSclMax;
MTPBase.RpmUnit := RpmUnit;
MTPBase.RpmMin := RpmMin;
MTPBase.RpmMax := RpmMax;
MTPBase.RpmRbk := RpmRbk;
MTPBase.RevFbkCalc := RevFbkCalc;
MTPBase.RevFbk := RevFbk;
MTPBase.FwdFbkCalc := FwdFbkCalc;
MTPBase.FwdFbk := FwdFbk;
MTPBase.Trip := Trip;
MTPBase.ResetAut := ResetAut;
MTPBase.MonSafePos := MonSafePos;
MTPBase.MonStatTi := MonStatTi;
MTPBase.MonDynTi := MonDynTi;
                
            
        
END_FUNCTION_BLOCK
